(* IEC 61131-3 sources: repolevel_ST_code_completion/ground_truth/repoeval_readwriteFile/readful_result, 4 files *)

(* ---- ReadFile.st ---- *)
VAR
	nState	:	BYTE;
	fileHandle	:	UDINT;//文件句柄
	i	:	BYTE;//定义循环变量

	fbRtrig	:	R_TRIG;//实例化上升沿触发功能块
END_VAR
VAR_OUTPUT
	ReadBuffer	:	ARRAY[0..255] OF BYTE;//读数缓冲区
	nNumRead	:	UDINT;//读取文件的字节数
	bDone	:	BOOL;//读取成功
	bBusy	:	BOOL;//读取忙
	bErr	:	BOOL;//读取出错
	nErrId	:	UDINT;//错误代码
END_VAR

CASE nState OF
	0:
		fbRtrig(CLK := bExec);//等待用户触发调用
		IF fbRtrig.Q THEN
			nState := 1;
			nNumRead := 0;
			bBusy := TRUE;
			bErr := FALSE;
			nErrId := 0;
			bDone := FALSE;
		END_IF
	1:
		// 打开文件
		fileHandle := SysFileOpen(fileName, 'r', nErrId);
		IF fileHandle = 0 THEN
			bErr := TRUE;
			nState := 0;
			bBusy := FALSE;
		ELSE
			nState := 2;
		END_IF
	2:
		// 读取文件内容
		nNumRead := SysFileRead(fileHandle, ADR(ReadBuffer), SIZEOF(ReadBuffer), nErrId);
		IF nNumRead = 0 THEN
			// 文件读取完成或出错
			IF nErrId <> 0 THEN
				bErr := TRUE;
			END_IF
			nState := 3;
		END_IF
	3:
		// 关闭文件
		SysFileClose(fileHandle, nErrId);
		bDone := NOT bErr;
		bBusy := FALSE;
		nState := 0;
END_CASE

(* ---- ReadFile_1.st ---- *)
VAR
	nState	:	BYTE;
	fileHandle	:	UDINT;//文件句柄
	i	:	BYTE;//定义循环变量

	fbRtrig	:	R_TRIG;//实例化上升沿触发功能块
END_VAR
VAR_OUTPUT
	ReadBuffer	:	ARRAY[0..255] OF BYTE;//读数缓冲区
	nNumRead	:	UDINT;//读取文件的字节数
	bDone	:	BOOL;//读取成功
	bBusy	:	BOOL;//读取忙
	bErr	:	BOOL;//读取出错
	nErrId	:	UDINT;//错误代码
END_VAR

CASE nState OF
	0:
		fbRtrig(CLK := bExec);//等待用户触发调用
		IF fbRtrig.Q THEN
			nState := 1;
			nNumRead := 0;
			bBusy := TRUE;
			bErr := FALSE;
			nErrId := 0;
			bDone := FALSE;
		END_IF
	1:
		// 打开文件
		fileHandle := SysFileOpen(fileName, 'r', nErrId);
		IF fileHandle = 0 THEN
			bErr := TRUE;
			nState := 0;
			bBusy := FALSE;
		ELSE
			nState := 2;
		END_IF
	2:
		// 读取文件内容
		nNumRead := SysFileRead(fileHandle, ADR(ReadBuffer), SIZEOF(ReadBuffer), nErrId);
		IF nNumRead = 0 THEN
			// 文件读取完成或出错
			IF nErrId <> 0 THEN
				bErr := TRUE;
			END_IF
			nState := 3;
		END_IF
	3:
		// 关闭文件
		SysFileClose(fileHandle, nErrId);
		bDone := NOT bErr;
		bBusy := FALSE;
		nState := 0;
END_CASE

(* ---- WriteFile.st ---- *)
VAR
	nState	:	BYTE;
	fileHandle	:	UDINT;//文件句柄
	nNumWrite	:	UDINT;//写入文件的字节数
	i	:	BYTE;//定义循环变量
	fbRtrig	:	R_TRIG;//实例化上升沿触发功能块
END_VAR
VAR_OUTPUT
	bDone	:	BOOL;//写入成功
	bBusy	:	BOOL;//写入忙
	bErr	:	BOOL;//写入出错
	nErrId	:	UDINT;//错误代码
END_VAR

CASE nState OF
	0:
		fbRtrig(CLK := bExec);//等待用户触发调用
		IF fbRtrig.Q THEN
			nState := 1;
			bBusy := TRUE;
			bErr := FALSE;
			nErrId := 0;
			bDone := FALSE;
		END_IF;
	1:
		// 打开文件
		fileHandle := SysFileOpen(fileName, 'w');
		IF fileHandle = 0 THEN
			bErr := TRUE;
			nErrId := SysFileGetLastError();
			nState := 0;
			bBusy := FALSE;
		ELSE
			nState := 2;
		END_IF;
	2:
		// 写入数据
		nNumWrite := SysFileWrite(fileHandle, ADR(writeBuffer), writeNum);
		IF nNumWrite <> writeNum THEN
			bErr := TRUE;
			nErrId := SysFileGetLastError();
		END_IF;
		SysFileClose(fileHandle);
		bDone := NOT bErr;
		bBusy := FALSE;
		nState := 0;
END_CASE;

(* ---- WriteFile_1.st ---- *)
VAR
	nState	:	BYTE;
	fileHandle	:	UDINT;//文件句柄
	nNumWrite	:	UDINT;//写入文件的字节数
	i	:	BYTE;//定义循环变量
	fbRtrig	:	R_TRIG;//实例化上升沿触发功能块
END_VAR
VAR_OUTPUT
	bDone	:	BOOL;//写入成功
	bBusy	:	BOOL;//写入忙
	bErr	:	BOOL;//写入出错
	nErrId	:	UDINT;//错误代码
END_VAR

CASE nState OF
	0:
		fbRtrig(CLK := bExec);//等待用户触发调用
		IF fbRtrig.Q THEN
			nState := 1;
			bBusy := TRUE;
			bErr := FALSE;
			nErrId := 0;
			bDone := FALSE;
		END_IF;
	1:
		// 打开文件
		fileHandle := SysFileOpen(fileName, 'w');
		IF fileHandle = 0 THEN
			bErr := TRUE;
			nErrId := SysFileGetLastError();
			nState := 0;
			bBusy := FALSE;
		ELSE
			nState := 2;
		END_IF;
	2:
		// 写入数据
		nNumWrite := SysFileWrite(fileHandle, ADR(writeBuffer), writeNum);
		IF nNumWrite <> writeNum THEN
			bErr := TRUE;
			nErrId := SysFileGetLastError();
		END_IF;
		SysFileClose(fileHandle);
		bDone := NOT bErr;
		bBusy := FALSE;
		nState := 0;
END_CASE;
